(* IEC 61131-3 sources: 2026_Projet_YGO_ExcavatriceDragage/TOOLS/TEST_AUTO_CI/RESULTS/_TROUBLESHOOTING/DSH01_T255D_FDC_BAS/tests, 3 files *)

(* ---- test_t255d_fdc_bas_exploratory.st ---- *)
(* =======================================================================
   T255-D — Reproduction exploratoire : AnyFault allume, bandeau muet
   -----------------------------------------------------------------------
   HORS CI OFFICIEL (dossier _TROUBLESHOOTING jetable, skill troubleshooting
   section 4ter). But : reproduire par EXECUTION le symptome terrain MES avant
   tout correctif. Un TEST par preuve (le harnais consigne un seul echec par test).

   Canal : harnais d'integration officiel FB_TestHarness_PRG_07 (PRG_07_Supervision),
   qui execute le formateur de bandeau avec les bus d'entree PRG_02/03/04/05.
   La cause est injectee par WinchData.WinchM1Safety / WinchM2Safety, exactement
   comme PRG_04 la publie.

   Fait de code vise :
     FB_Safety_Winch.st:318-325   instCauses[6] (bit6 = 16#0040), cause LIVE
                                  'Limite basse cable atteinte'
     FB_FaultCore.st:49-57        Error := (ErrorId <> 0)  -> vue LIVE
     FB_WinchStateProjection.st:236-237
                                  Safety.Error agrege les deux FBs,
                                  Safety.ErrorId = securite uniquement
     PRG_07_Supervision.st:537-547  AnyFaultActive agrege Safety.Error
     FB_Hmi_BannerFormatter.st:812-849   carrousel : bit6 NON decode
     FB_Hmi_BannerFormatter.st:648-658   seul libelle, sous commande descente

   Preuves attendues sur le code du 2026-09-20 (aucun correctif) :
     -A1  ROUGE : aucun canal du bandeau n'expose la cause (carrousel vide,
                  SpecialCondition vide) alors que la cause allume AnyFaultActive
     -A2  ROUGE : le texte daction reste le rappel joystick generique
   Apres correctif : les 4 tests doivent etre VERTS.
   ======================================================================= *)

SETUP
VAR
    PRG07 : FB_TestHarness_PRG_07;
    AcqData : ST_AcquisitionInterPrg;
    ModesAuth : ST_Modes_Autorisations;
    WinchData : ST_WinchInterPrg;
    TranslationData : ST_TranslationInterPrg;
END_VAR

// Pas de boot long : au dela de 1,5 s les filtres anti-bagotement invalideraient le
// reseau (le harnais ne cable pas Network), ce qui masquerait la cause visee par une
// alarme parente de module E/S. TonBootInhibit (4 s) protege les 4 tests.
ModesAuth.Mode := E_Mode.MAINT_N1;
ModesAuth.JoystickWinchSelectArbitrated := 0;   // treuils couples -> CurrentDirection = WinchBothMotionDirection = 0
AcqData.Joystick.DeadmanArmed := FALSE;         // situation terrain : joystick relache
AcqData.Joystick.AtNeutralXY := TRUE;
END_SETUP

TEST 'T255D-REPRO-M1-A1 butte basse cable M1 : aucun canal du bandeau nexpose la cause active'
    WinchData.WinchM1Safety.Error := TRUE;           (* vu par AnyFaultActive *)
    WinchData.WinchM1Safety.ErrorId := 16#0040;      (* bit6 = limite basse cable, vue LIVE *)
    WinchData.WinchM1Safety.CableLimitDescent := TRUE;
    WinchData.WinchM1Safety.DescendPermit := FALSE;  (* interlock : descente interdite *)
    WinchData.WinchM1Safety.AscentPermit := TRUE;    (* remontee autorisee *)
    WinchData.WinchM2Safety.AscentPermit := TRUE;

    PRG07(AcqData := AcqData, ModesAuth := ModesAuth, WinchData := WinchData,
          TranslationData := TranslationData, EmergencyChainClosed := TRUE,
          PowerContactorEngaged := TRUE, PowerCutOffActive := FALSE, BtnResetMachine := FALSE);
    ADVANCE_TIME(600000000);
    PRG07(AcqData := AcqData, ModesAuth := ModesAuth, WinchData := WinchData,
          TranslationData := TranslationData, EmergencyChainClosed := TRUE,
          PowerContactorEngaged := TRUE, PowerCutOffActive := FALSE, BtnResetMachine := FALSE);

    ASSERT_TRUE(PRG07.Banner.AlarmBanner.HasAlarm OR PRG07.Banner.SpecialConditionText <> '',
                '[T255D-A1] cause limite basse cable M1 active : aucun canal du bandeau ne lexpose');
END_TEST

TEST 'T255D-REPRO-M1-A2 butte basse cable M1 : le texte daction ne nomme pas la cause'
    WinchData.WinchM1Safety.Error := TRUE;
    WinchData.WinchM1Safety.ErrorId := 16#0040;
    WinchData.WinchM1Safety.CableLimitDescent := TRUE;
    WinchData.WinchM1Safety.DescendPermit := FALSE;
    WinchData.WinchM1Safety.AscentPermit := TRUE;
    WinchData.WinchM2Safety.AscentPermit := TRUE;

    PRG07(AcqData := AcqData, ModesAuth := ModesAuth, WinchData := WinchData,
          TranslationData := TranslationData, EmergencyChainClosed := TRUE,
          PowerContactorEngaged := TRUE, PowerCutOffActive := FALSE, BtnResetMachine := FALSE);
    ADVANCE_TIME(600000000);
    PRG07(AcqData := AcqData, ModesAuth := ModesAuth, WinchData := WinchData,
          TranslationData := TranslationData, EmergencyChainClosed := TRUE,
          PowerContactorEngaged := TRUE, PowerCutOffActive := FALSE, BtnResetMachine := FALSE);

    ASSERT_NEQ(PRG07.Banner.OperatorActionText, '[JOYSTICK] Appuyer homme-mort au neutre',
               '[T255D-A2] la cause limite basse cable M1 doit etre nommee dans laction');
END_TEST

TEST 'T255D-REPRO-M2-A1 butte basse cable M2 : aucun canal du bandeau nexpose la cause active'
    WinchData.WinchM2Safety.Error := TRUE;
    WinchData.WinchM2Safety.ErrorId := 16#0040;
    WinchData.WinchM2Safety.CableLimitDescent := TRUE;
    WinchData.WinchM2Safety.DescendPermit := FALSE;
    WinchData.WinchM2Safety.AscentPermit := TRUE;
    WinchData.WinchM1Safety.AscentPermit := TRUE;

    PRG07(AcqData := AcqData, ModesAuth := ModesAuth, WinchData := WinchData,
          TranslationData := TranslationData, EmergencyChainClosed := TRUE,
          PowerContactorEngaged := TRUE, PowerCutOffActive := FALSE, BtnResetMachine := FALSE);
    ADVANCE_TIME(600000000);
    PRG07(AcqData := AcqData, ModesAuth := ModesAuth, WinchData := WinchData,
          TranslationData := TranslationData, EmergencyChainClosed := TRUE,
          PowerContactorEngaged := TRUE, PowerCutOffActive := FALSE, BtnResetMachine := FALSE);

    ASSERT_TRUE(PRG07.Banner.AlarmBanner.HasAlarm OR PRG07.Banner.SpecialConditionText <> '',
                '[T255D-A1] cause limite basse cable M2 active : aucun canal du bandeau ne lexpose');
END_TEST

TEST 'T255D-REPRO-M2-A2 butte basse cable M2 : le texte daction ne nomme pas la cause'
    WinchData.WinchM2Safety.Error := TRUE;
    WinchData.WinchM2Safety.ErrorId := 16#0040;
    WinchData.WinchM2Safety.CableLimitDescent := TRUE;
    WinchData.WinchM2Safety.DescendPermit := FALSE;
    WinchData.WinchM2Safety.AscentPermit := TRUE;
    WinchData.WinchM1Safety.AscentPermit := TRUE;

    PRG07(AcqData := AcqData, ModesAuth := ModesAuth, WinchData := WinchData,
          TranslationData := TranslationData, EmergencyChainClosed := TRUE,
          PowerContactorEngaged := TRUE, PowerCutOffActive := FALSE, BtnResetMachine := FALSE);
    ADVANCE_TIME(600000000);
    PRG07(AcqData := AcqData, ModesAuth := ModesAuth, WinchData := WinchData,
          TranslationData := TranslationData, EmergencyChainClosed := TRUE,
          PowerContactorEngaged := TRUE, PowerCutOffActive := FALSE, BtnResetMachine := FALSE);

    ASSERT_NEQ(PRG07.Banner.OperatorActionText, '[JOYSTICK] Appuyer homme-mort au neutre',
               '[T255D-A2] la cause limite basse cable M2 doit etre nommee dans laction');
END_TEST

(* ---- test_t255d_fdc_bas_hypotheses.st ---- *)
(* =======================================================================
   T255-D — Reproduction exploratoire : mecanisme (A) du brief CC01
   -----------------------------------------------------------------------
   HORS CI OFFICIEL (dossier _TROUBLESHOOTING jetable, skill troubleshooting
   section 4ter). Cas FB_Hmi_BannerFormatter avec registre ephemere : les 13
   sources absentes du dossier 5_ASSISTANCE_DRAGAGE sont retirees et
   E_CycleDepthStopMode.st est ajoutee (entree officielle cassee, decision D4).

   Question mesuree : un defaut LATCHE et BLOQUANT, actif, disparait-il du
   carrousel quand un flag de validite materielle passe a FALSE (mecanisme A) ?

   MecaB (bit8 = 16#0100, Latching := TRUE — FB_Safety_Winch.st:339-350) est un
   defaut bloquant : il entre dans CausesSafeStop et CausesPowerCutOff.
   Son entree carrousel est gardee par EncM1Valid (FB_Hmi_BannerFormatter.st:829).

   A1 : materiel sain            -> la cause doit etre visible
   A2 : meme cause + codeur M1 perdu -> la cause disparait, remplacee par le parent ECAT
   ======================================================================= *)

SETUP
VAR
    FB_Banner : FB_Hmi_BannerFormatter;
    WinchM1Safety : ST_SafetyWinch;
    WinchM2Safety : ST_SafetyWinch;
    TranslationSafety : ST_SafetyTranslation;
    NetDiag : ST_NetworkDiagHMI;
END_VAR

NetDiag.InputModules.LocalDigitalIoOk := TRUE;
NetDiag.InputModules.Vh0800EndOk := TRUE;
NetDiag.InputModules.Vh0808EtpOk := TRUE;
NetDiag.InputModules.Vh0008ErOk := TRUE;
NetDiag.InputModules.Vh0008Er1Ok := TRUE;
NetDiag.BusCanOpen.Operational := TRUE;
NetDiag.Joystick.Operational := TRUE;
NetDiag.BusEthercat.Operational := TRUE;
NetDiag.EncoderM1.Operational := TRUE;
NetDiag.EncoderM2.Operational := TRUE;
NetDiag.VariateurM3.Operational := TRUE;
END_SETUP

TEST 'T255D-HYP-A1 MecaB latche et bloquant, materiel sain : la cause est visible'
    FB_Banner(Enable := TRUE, CurrentMode := E_Mode.MAINT_N1,
              EmergencyChainClosed := TRUE, PowerContactorEngaged := TRUE,
              WinchM1Safety := WinchM1Safety, WinchM2Safety := WinchM2Safety,
              Network := NetDiag);
    ADVANCE_TIME(5000000000);

    WinchM1Safety.Error := TRUE;
    WinchM1Safety.ErrorId := 16#0100;      (* bit8 = MecaB *)
    WinchM1Safety.LatchedId := 16#0100;
    WinchM1Safety.ErrorMecaB := TRUE;

    FB_Banner(Enable := TRUE, CurrentMode := E_Mode.MAINT_N1,
              EmergencyChainClosed := TRUE, PowerContactorEngaged := TRUE,
              WinchM1Safety := WinchM1Safety, WinchM2Safety := WinchM2Safety,
              Network := NetDiag);

    ASSERT_TRUE(FB_Banner.Banner.AlarmBanner.HasAlarm,
                '[T255D-HYP-A1] materiel sain : le defaut bloquant MecaB doit etre au carrousel');
    ASSERT_EQ(FB_Banner.Banner.AlarmBanner.Text,
              '1/1 [M1] ErrorID:09 - MecaB - arret non confirme apres stop',
              '[T255D-HYP-A1] libelle attendu du defaut MecaB');
END_TEST

TEST 'T255D-HYP-A2 meme defaut + codeur M1 perdu : cause BLOQUANTE masquee par le parent ECAT'
    FB_Banner(Enable := TRUE, CurrentMode := E_Mode.MAINT_N1,
              EmergencyChainClosed := TRUE, PowerContactorEngaged := TRUE,
              WinchM1Safety := WinchM1Safety, WinchM2Safety := WinchM2Safety,
              Network := NetDiag);
    ADVANCE_TIME(5000000000);

    WinchM1Safety.Error := TRUE;
    WinchM1Safety.ErrorId := 16#0100;      (* bit8 = MecaB, toujours ACTIF *)
    WinchM1Safety.LatchedId := 16#0100;
    WinchM1Safety.ErrorMecaB := TRUE;
    NetDiag.EncoderM1.Operational := FALSE; (* EncM1Valid passe a FALSE *)

    FB_Banner(Enable := TRUE, CurrentMode := E_Mode.MAINT_N1,
              EmergencyChainClosed := TRUE, PowerContactorEngaged := TRUE,
              WinchM1Safety := WinchM1Safety, WinchM2Safety := WinchM2Safety,
              Network := NetDiag);

    ASSERT_TRUE(FB_Banner.Banner.AlarmBanner.HasAlarm,
                '[T255D-HYP-A2] le parent materiel reste affiche : le bandeau nest pas vide');
    ASSERT_EQ(FB_Banner.Banner.AlarmBanner.Count, 1,
              '[T255D-HYP-A2] une seule alarme : le parent ECAT seulement');
    ASSERT_EQ(FB_Banner.Banner.AlarmBanner.Text,
              '1/1 [M1] Codeur absolu COD1 non detecte (ECAT)',
              '[T255D-HYP-A2] la cause BLOQUANTE MecaB est absente : masquee par EncM1Valid');
END_TEST

(* ---- test_t255d_fdc_bas_producer.st ---- *)
(* =======================================================================
   T255-D — Reproduction exploratoire, PRODUCTEUR : FB_Safety_Winch
   -----------------------------------------------------------------------
   HORS CI OFFICIEL (dossier _TROUBLESHOOTING jetable, skill troubleshooting
   section 4ter).

   But : trancher par EXECUTION la semantique de la vue publiee par le socle de
   defaut, sur la seule cause « limite basse cable atteinte » (instCauses[6],
   bit6 = 16#0040, Latching := FALSE — FB_Safety_Winch.st:318-325).

   Question tranchee : une limite basse cable SEULE allume-t-elle Fault.Error
   (vue LIVE) sans aucun defaut latche ?

     FB_FaultCore.st:49-57   Fault.ErrorId := bitfield des Causes[i].Active
                             Fault.Error := (Fault.ErrorId <> 0)   <- vue LIVE
     FB_FaultCore.st:60-81   Latched / LatchedId = vue LATCHEE (Latching=TRUE seulement)

   Attendu : Error = TRUE, ErrorId = 16#0040, Latched = FALSE.
   ======================================================================= *)

SETUP
VAR
    SafetyW : FB_Safety_Winch;
END_VAR
END_SETUP

TEST 'T255D-PROD-1 limite basse cable seule : Fault.Error (vue LIVE) est allume'
    SafetyW(Enable := TRUE, Reset := FALSE, Mode := E_Mode.MAINT_N1,
            SyncEnable := FALSE, CrossCheckEnable := FALSE,
            PowerContactorEngaged := TRUE,
            JoystickOnline := TRUE, JoystickOperational := TRUE, HeartbeatIhmOk := TRUE,
            EncoderAvailable := TRUE,
            ThermalFeedback := FALSE, BrakeThermalFeedback := FALSE,
            SlackCableDetected := FALSE, PhaseRotationOk := TRUE,
            TopPositionSensor := TRUE,
            FwdRevSpeedFeedbackOff := TRUE, BrakeFeedback := FALSE,
            JoystickYNeutral := TRUE, BenneHoldStillActive := FALSE, BenneBusy := FALSE,
            OtherWinchInhibited := FALSE,
            InReferencingMode := FALSE,
            CablePosM := -50.1, CfgCableLimitDescentM := -50.0,
            LimitLegalReached := FALSE, Homed := TRUE, HomingSuspect := FALSE, TopLimitM := 7.5,
            ReqAscent := FALSE, ReqDescend := FALSE, MovementCommanded := FALSE,
            ExpectedOtherWinchPosM := -50.1,
            MeasuredSpeedValid := TRUE, MeasuredSpeedMps := 0.0, MeasuredSpeedSignedMps := 0.0,
            SpeedBandMaxMps := 3.0,
            BypassGlobal := FALSE, BypassSafety := FALSE, BypassProcess := FALSE,
            BypassCableLimitSwitch := FALSE, BypassTopLimitSwitch := FALSE,
            BypassMecaA := FALSE, BypassMecaB := FALSE, BypassMecaC := FALSE,
            BypassMecaD := FALSE, BypassMecaE := FALSE, BypassOperatorComm := FALSE,
            BypassPhaseRotation := FALSE, BypassBrakeThermal := FALSE,
            BypassMotorThermal := FALSE);

    ASSERT_TRUE(SafetyW.Fault.Error,
                '[T255D-PROD-1] une limite basse cable seule doit allumer la vue LIVE Fault.Error');
END_TEST

TEST 'T255D-PROD-2 limite basse cable seule : ErrorId = 16#0040 et AUCUN defaut latche'
    SafetyW(Enable := TRUE, Reset := FALSE, Mode := E_Mode.MAINT_N1,
            SyncEnable := FALSE, CrossCheckEnable := FALSE,
            PowerContactorEngaged := TRUE,
            JoystickOnline := TRUE, JoystickOperational := TRUE, HeartbeatIhmOk := TRUE,
            EncoderAvailable := TRUE,
            ThermalFeedback := FALSE, BrakeThermalFeedback := FALSE,
            SlackCableDetected := FALSE, PhaseRotationOk := TRUE,
            TopPositionSensor := TRUE,
            FwdRevSpeedFeedbackOff := TRUE, BrakeFeedback := FALSE,
            JoystickYNeutral := TRUE, BenneHoldStillActive := FALSE, BenneBusy := FALSE,
            OtherWinchInhibited := FALSE,
            InReferencingMode := FALSE,
            CablePosM := -50.1, CfgCableLimitDescentM := -50.0,
            LimitLegalReached := FALSE, Homed := TRUE, HomingSuspect := FALSE, TopLimitM := 7.5,
            ReqAscent := FALSE, ReqDescend := FALSE, MovementCommanded := FALSE,
            ExpectedOtherWinchPosM := -50.1,
            MeasuredSpeedValid := TRUE, MeasuredSpeedMps := 0.0, MeasuredSpeedSignedMps := 0.0,
            SpeedBandMaxMps := 3.0,
            BypassGlobal := FALSE, BypassSafety := FALSE, BypassProcess := FALSE,
            BypassCableLimitSwitch := FALSE, BypassTopLimitSwitch := FALSE,
            BypassMecaA := FALSE, BypassMecaB := FALSE, BypassMecaC := FALSE,
            BypassMecaD := FALSE, BypassMecaE := FALSE, BypassOperatorComm := FALSE,
            BypassPhaseRotation := FALSE, BypassBrakeThermal := FALSE,
            BypassMotorThermal := FALSE);

    ASSERT_EQ(SafetyW.Fault.ErrorId, 16#0040,
              '[T255D-PROD-2] ErrorId attendu = bit6 seul (limite basse cable)');
    ASSERT_FALSE(SafetyW.Fault.Latched,
                 '[T255D-PROD-2] aucun defaut latche ne doit etre present : Latched reste FALSE');
END_TEST
